Staubli VAL3: Pick.pgx

program pick(point pPosition, tool tTool, mdesc mApproach, mdesc mTarget)
  local point pOffset
begin

  // Función para coger la pieza desde el punto donde se alimenta
  pOffset=appro(pPosition,{0,0,-50,0,0,0})
  // Se aproxima al destino
  movej(pOffset,tTool,mApproach)
  movel(pPosition,tTool,mTarget)
  close(tTool)
  movel(pOffset,tTool,mTarget)

end
